FUNCTION_BLOCK BACnetBinaryOutput (* Service Interface Function Block Type *)
  (* Standard: 61499-2 *)
  (* Version 1.0, 2020-03-03, root *)
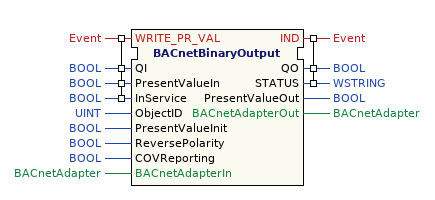
  EVENT_INPUT
    WRITE_PR_VAL WITH PresentValueIn, QI, InService; (* Service Initialization *)
  END_EVENT
  EVENT_OUTPUT
    IND WITH QO, STATUS; (* Indication *)
  END_EVENT
  VAR_INPUT
    QI : BOOL; (* Event Input Qualifier *)
    PresentValueIn : BOOL;
    InService : BOOL;
    ObjectID : UINT;
    PresentValueInit : BOOL;
    ReversePolarity : BOOL;
    COVReporting : BOOL;
  END_VAR
  VAR_OUTPUT
    QO : BOOL; (* Event Output Qualifier *)
    STATUS : WSTRING;
    PresentValueOut : BOOL;
  END_VAR
  SOCKETS
    BACnetAdapterIn : BACnetAdapter;
  END_SOCKETS
  PLUGS
    BACnetAdapterOut : BACnetAdapter;
  END_PLUGS
END_FUNCTION_BLOCK
